INTERFACE ITF_Color

METHOD applyColor : STRING
END_METHOD

END_INTERFACE

(* stored: Version 1.1.0.1, ProductVersion 3.1.4024.12
   Itf ITF_Color: Id {8dedefbb-c13c-4893-aa9f-6b9ec5c7c489}
   Method applyColor: Id {915f56a5-5524-43be-b073-8672042dbc3d} *)
